(* CODESYS project Soru_1.project
   Title: Adsız2
   Version: 0.0.0.0
   Author: Enes

Project tree, tasks and I/O mapping:
  MyController : TM241C24T/U, Schneider Electric, order no. TM241C24T/U, version 4.0.6.18
    application Application
      task MAST (cyclic, interval 20 ms, priority 15, watchdog 100 ms x 1) calls POU
      global variables GVL
      program POU [LD]
    DI : Digital Inputs, Schneider Electric, version 4.0.6.18
        input  iwDI_IW0 : WORD  // IW0
        input  ibDI_IB1 : BYTE  // IB1
    DQ : Digital Outputs, Schneider Electric, version 4.0.6.18
        output qwDQ_QW0 : WORD  // QW0
        output qbDQ_QB1 : BYTE  // QB1
    Counters : Counters, Schneider Electric, version 4.0.6.18
    Pulse_Generators : Pulse Generators, Schneider Electric, version 4.0.6.18
    Cartridge_1 : Cartridge, Schneider Electric, version 4.0.6.18
    IO_Bus : IO bus - TM3, Schneider Electric, version 4.0.6.18
    COM_Bus : COM bus, Schneider Electric, version 4.0.6.18
    Serial_Line_1 : Serial line, Schneider Electric, version 4.0.6.18
      SoMachine_Network_Manager : SoMachine-Network Manager, Schneider Electric, version 4.0.0.2
    Serial_Line_2 : Serial line, Schneider Electric, version 4.0.6.18
      Modbus_Manager : Modbus Manager, Schneider Electric, version 4.0.0.2
*)

// MyController/Application/GVL
VAR_GLOBAL
END_VAR

// MyController/Application/POU
PROGRAM POU
VAR
	
	M0: BOOL;
	Baslat: BOOL;
	Durdur: BOOL;
	Motor: BOOL;
	Timer1: TON;
	Timer2: TON;
END_VAR

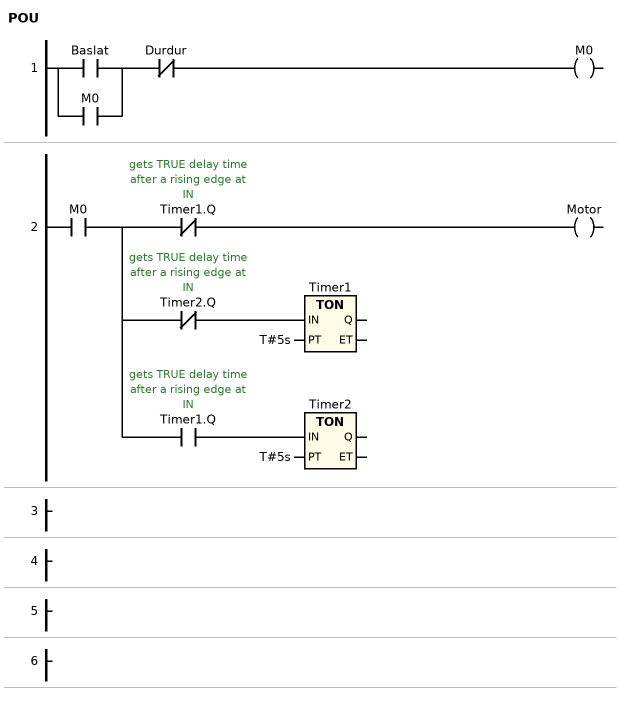
// NETWORK 1
M0 := (Baslat OR M0) AND NOT Durdur;

// NETWORK 2
//   Timer1.Q: gets TRUE delay time after a rising edge at IN
//   Timer2.Q: gets TRUE delay time after a rising edge at IN
Motor := M0 AND NOT Timer1.Q;
Timer1(IN := M0 AND NOT Timer2.Q, PT := T#5s); // TON
Timer2(IN := M0 AND Timer1.Q, PT := T#5s); // TON

// NETWORK 3

// NETWORK 4

// NETWORK 5

// NETWORK 6

END_PROGRAM
